(* PLC project Unnamed, Unknown Unnamed 1 *)
(* stored: creationDateTime 2025-03-11T14:10:47, modificationDateTime 2025-03-11T14:53:34 *)

PROGRAM main
  VAR
    St0 : BOOL := 1;
    St1 : BOOL := 0;
    St2 : BOOL := 0;
    St3 : BOOL := 0;
    St4 : BOOL := 0;
    St5 : BOOL := 0;
    BoxBut : BOOL := 0;
    StartBut : BOOL := 0;
    My_Time : BOOL := 0;
    BB : BOOL := 0;
    BB2 : BOOL := 0;
    Motor : BOOL := 0;
  END_VAR

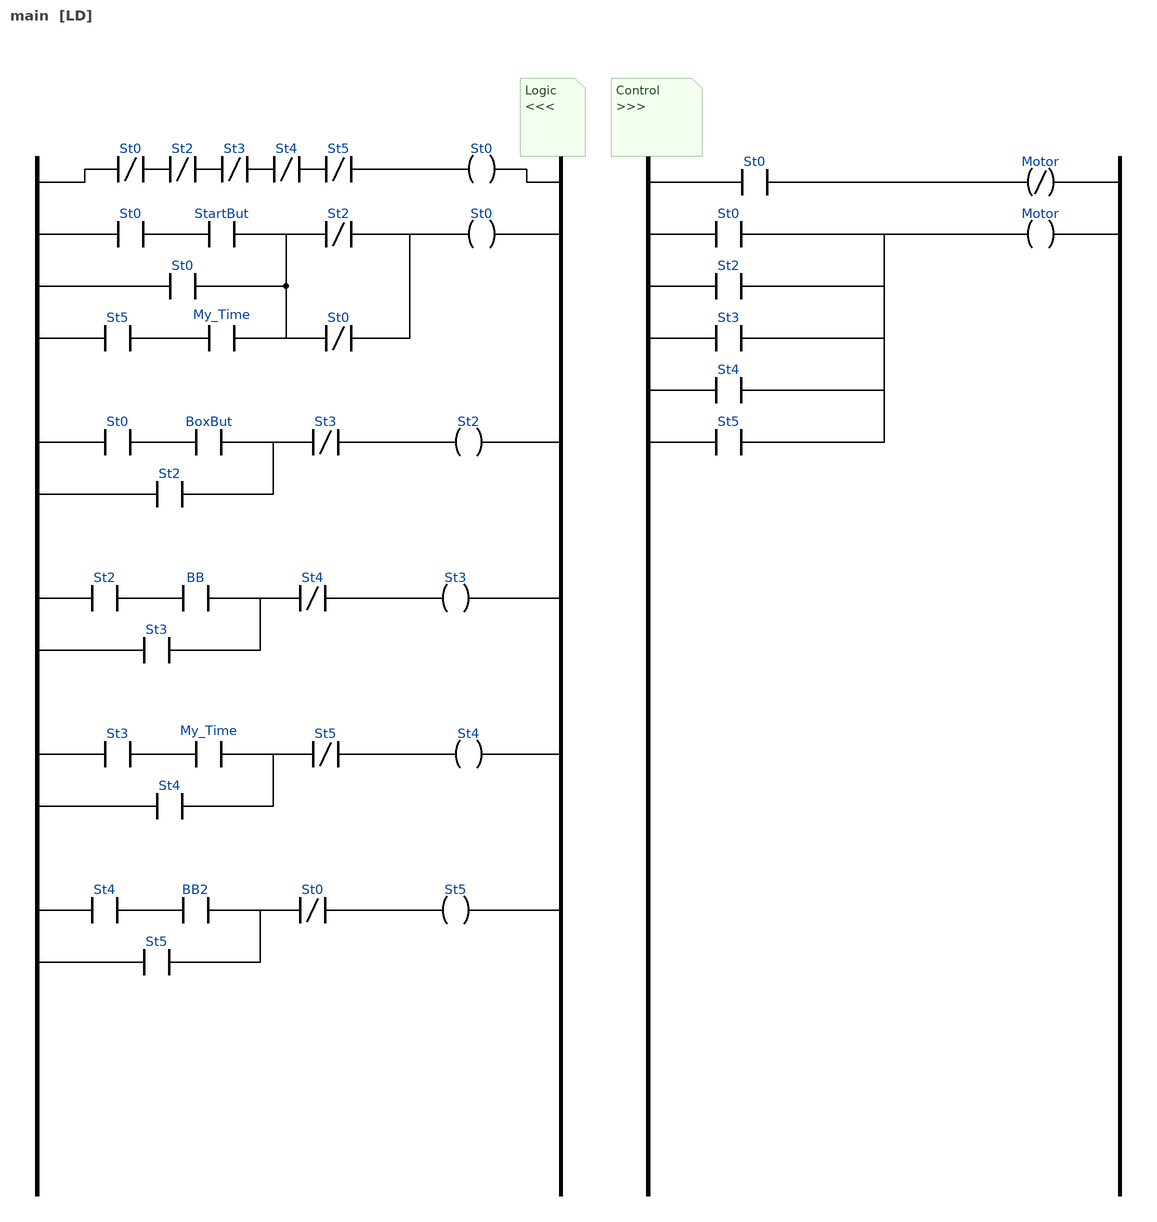
(* LD diagram, written out as Structured Text *)
(* Logic
<<< *)
(* Control
>>> *)
St0 := St0 AND NOT St2 OR (St5 AND My_Time OR St0) AND NOT St0;
St0 := NOT St0 AND NOT St2 AND NOT St3 AND NOT St4 AND NOT St5;
St2 := (St0 AND BoxBut OR St2) AND NOT St3;
St3 := (St2 AND BB OR St3) AND NOT St4;
St4 := (St3 AND My_Time OR St4) AND NOT St5;
St5 := (St4 AND BB2 OR St5) AND NOT St0;
Motor := NOT St0;
Motor := St0 OR St2 OR St3 OR St4 OR St5;
END_PROGRAM

CONFIGURATION Config0
  RESOURCE Res0 ON PLC
    TASK task0(INTERVAL := T#20ms, PRIORITY := 0);
    PROGRAM instance0 WITH task0 : main;
  END_RESOURCE
END_CONFIGURATION
